// TIA Portal V20 export
ORGANIZATION_BLOCK "Main"   // OB1, LAD, ProgramCycle
TITLE = "Main Program Sweep (Cycle)"
{ S7_Optimized_Access := 'TRUE' }
// stored: SetENOAutomatically false
   VAR_INPUT
      Initial_Call : Bool;   // Initial call of this OB
      Remanence : Bool;   // =True, if remanent data are available
   END_VAR
BEGIN

REGION Network 1
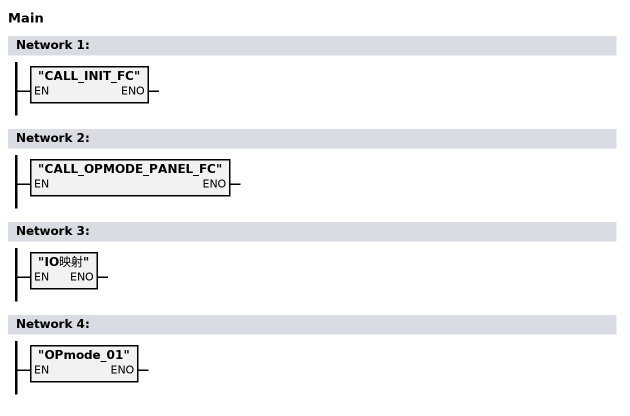
   RUNG wire#powerrail
      "CALL_INIT_FC"()
   END_RUNG
   // the same network as SCL:
   "CALL_INIT_FC"();
END_REGION

REGION Network 2
   RUNG wire#powerrail
      "CALL_OPMODE_PANEL_FC"()
   END_RUNG
   // the same network as SCL:
   "CALL_OPMODE_PANEL_FC"();
END_REGION

REGION Network 3
   RUNG wire#powerrail
      "IO映射"()
   END_RUNG
   // the same network as SCL:
   "IO映射"();
END_REGION

REGION Network 4
   RUNG wire#powerrail
      "OPmode_01"()
   END_RUNG
   // the same network as SCL:
   "OPmode_01"();
END_REGION
END_ORGANIZATION_BLOCK
